TYPE st_PlateHookStationMove :
STRUCT
	PlateHookPoint		: E_PlateHookPoint;
	Handshake			: ST_HandshakeBase;
END_STRUCT
END_TYPE

(* stored: Version 1.1.0.1, ProductVersion 3.1.4024.13
   DUT st_PlateHookStationMove: Id {7d587053-79c3-46cb-a236-d1a2b8009fac} *)
